TYPE ST_MoverDistance :
STRUCT
	nPositionIndex	: UDINT;
	fDistance		: LREAL;
END_STRUCT
END_TYPE

(* stored: Version 1.1.0.1, ProductVersion 3.1.4024.12
   DUT ST_MoverDistance: Id {e0f42923-d085-4707-af25-68f5d432a110} *)
